{attribute 'linkalways'}
{attribute 'hide_all_locals'}
FUNCTION_BLOCK ValueLtimeRead EXTENDS ValueBase IMPLEMENTS ValueRead
VAR
	thisValue : LTIME;
END_VAR

{attribute 'call_after_global_init_slot' := '1'}
{attribute 'call_after_online_change_slot' := '1'}
METHOD PROTECTED GetThisAnyType
VAR_INPUT
END_VAR
thisAnyType := ToAnyType(thisValue);
END_METHOD

METHOD GetAsType : BOOL
VAR_INPUT
	destination : __SYSTEM.AnyType;
END_VAR
GetAsType := ConvertAnyType(thisAnyType, destination);
END_METHOD

METHOD GetAsString : T_MaxString
VAR_INPUT
END_VAR
GetAsString := LTIME_TO_STRING(thisValue);
END_METHOD

METHOD Get : BOOL
VAR_INPUT
	destination : ANY;
END_VAR
Get := ConvertAnyType(thisAnyType, destination);
END_METHOD

METHOD FB_init : BOOL
VAR_INPUT
	bInitRetains : BOOL; // if TRUE, the retain variables are initialized (warm start / cold start)
	bInCopyCode : BOOL;  // if TRUE, the instance afterwards gets moved into the copy code (online change)
END_VAR
_ValueType := __SYSTEM.TYPE_CLASS.TYPE_LTIME;
END_METHOD

{attribute 'monitoring' := 'call'}
PROPERTY Value : LTIME
GET
Value := thisValue;
END_GET
END_PROPERTY

END_FUNCTION_BLOCK

(* stored: Version 1.1.0.1
   POU ValueLtimeRead: Id {d5630c5b-83ac-42b2-8de9-c978dc8c2b76}, SpecialFunc None
   Method GetThisAnyType: Id {3ba86803-5439-49f0-a3dc-93361baade50}
   Method GetAsType: Id {0a2b81fa-f829-4b9a-9de5-861215360bb7}
   Method GetAsString: Id {f8b042df-5cf3-4b97-b3b3-477d527db574}
   Method Get: Id {60db7ceb-0f5c-4c7a-8c69-35f100d08899}
   Method FB_init: Id {4ddcd487-49f2-46bd-8ce0-9db56f92d0ba}
   Property Value: Id {12091e06-6b10-4ab7-b193-d3eb7da8ddf6}
   Get Get: Id {7f5adf7e-1730-487c-adca-ffb370487367} *)
